PROGRAM prgEM
VAR
	fbKBusState		: FB_K_Bus_State;
	fbEM1			: FB_EM_Beckhoff_KL3403;

END_VAR


fbKBusState(	uiKBusState_OUT=> , 
				b_Kbus_notOk=> , 
				word_ErrorCount=> );
//The mapping OF THIS FUNCTION must be linked with the KL3403 in the E/A Part
// KEBA CS
fbEM1(
	bEnable:= true, 
	bChannel1Invers:= FALSE,				//Invert power data when transformer are mounted upside down
	bChannel2Invers:= FALSE,			
	bChannel3Invers:= FALSE,
	uiCurrentTransformerRatioL1:= 100, //Transformer ratio on the secondary side
	uiCurrentTransformerRatioL2:= 100, 
	uiCurrentTransformerRatioL3:= 100, 
	uiKBusState_IN:= fbKBusState.uiKBusState_OUT, 
	stDataEMPower=> , 
	stDataEMCounter=> , 
	stDataEMPowerRealTime=> , 
	stDataEMCounterRealTime=> , 
	diNrOfEM_OUT=> );

END_PROGRAM

(* stored: Version 1.1.0.1, ProductVersion 3.1.4024.12
   POU prgEM: Id {911a6298-93ee-4aec-855e-d2e16b0de8c7}, SpecialFunc None *)
